// TIA Portal V19 export
TYPE "lexchangetray_typeUnEmn_signalTM_Monitor"
// Type: Bool
// stored: Access Published
   STRUCT
      simulationed : Bool;   // Manual mode parameters for axis control interface
   END_STRUCT;
END_TYPE
